FUNCTION_BLOCK FB_TransferirPale_SFC
VAR_INPUT
	
	//Tiempo
	Tcheck: TIME := T#1S;	

	// SFC-Flags
	SFCPause: BOOL;
	SFCReset: BOOL;
	
	//Indicadores de sincronizacion
	Ack: BOOL:= TRUE;
	Execute: BOOL;
	
	//Entradas

	
END_VAR
VAR_OUTPUT
	//indicadores de sincronizacion
	Done: BOOL;
	Ready: BOOL;

	//Salidas
	Retenedor_pale_baja: BOOL;
	Activa_marcha_motor_cinta: BOOL;
	Separador_pale_sube: BOOL;
	
END_VAR
VAR
END_VAR

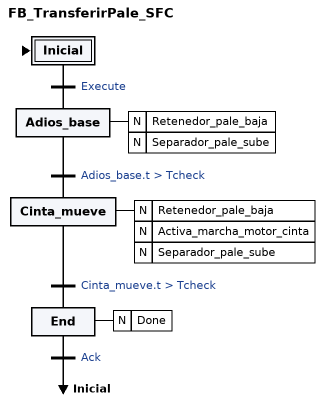
INITIAL_STEP Inicial:
END_STEP
TRANSITION FROM Inicial TO Adios_base
    := Execute;
END_TRANSITION
STEP Adios_base:
    Retenedor_pale_baja(N);
    Separador_pale_sube(N);
END_STEP
TRANSITION FROM Adios_base TO Cinta_mueve
    := Adios_base.t > Tcheck;
END_TRANSITION
STEP Cinta_mueve:
    Retenedor_pale_baja(N);
    Activa_marcha_motor_cinta(N);
    Separador_pale_sube(N);
END_STEP
TRANSITION FROM Cinta_mueve TO End
    := Cinta_mueve.t > Tcheck;
END_TRANSITION
STEP End:
    Done(N);
END_STEP
TRANSITION FROM End TO Inicial
    := Ack;
END_TRANSITION

END_FUNCTION_BLOCK

(* stored: Version 1.1.0.1, ProductVersion 3.1.4024.12
   POU FB_TransferirPale_SFC: Id {15ad5887-5800-4862-8886-2182498b3710}, SpecialFunc None *)
